(* IEC 61131-3 sources: repolevel_ST_code_completion/output/0127完整版本_带planner/repoeval_Builder_Application_RPI/readful_result_no_provide, 5 files *)

(* ---- ConcreteBuilder.st ---- *)
//This is the concrete builder class, reponsible for building the final product object
FUNCTION_BLOCK ConcreteBuilder
VAR_INPUT
END_VAR
VAR_OUTPUT
END_VAR
VAR
  isCompleted : BOOL := FALSE; // Indicates if the product construction is completed
  isValid : BOOL; // Indicates if the specifications are valid
  i : INT; // Loop variable
END_VAR

// Step 1: Initialize the product object
localProduct := Product(); // Add missing semicolon here
localProduct.Initialize();

// Step 2: Validate client specifications
isValid := TRUE;
FOR i := 1 TO 4 DO
    IF specifications[i] = '' THEN
        isValid := FALSE;
        EXIT;
    END_IF;
END_FOR;

// Step 3: Update product attributes based on specifications and director guidance
IF isValid THEN
    localProduct.Set_Main_Part(specifications[1]);
    localProduct.Set_Part1(specifications[2]);
    localProduct.Set_Part2(specifications[3]);
    localProduct.Set_Part3(specifications[4]);
END_IF;

// Step 4: Mark product as completed if valid
IF isValid THEN
    isCompleted := TRUE;
    localProduct.Mark_As_Completed();
END_IF;

// Step 5: Return the constructed product object
// Remove invalid RETURN statements to avoid syntax errors
IF isCompleted THEN
  RETURN; // Correctly use RETURN with no object
ELSE
  RETURN; // Correctly use RETURN with no object
END_IF;
END_FUNCTION_BLOCK

(* ---- Director.st ---- *)
VAR
    product : Product; // Local variable to store the final product object.
END_VAR

IF inputConcreteBuilder <> 0 THEN
    // Assign the input concrete builder to the Director's concreteBuilder field.
    THIS^.concreteBuilder := inputConcreteBuilder;

    // Step-by-step construction of the product using the concrete builder.
    THIS^.concreteBuilder.Set_Main_Part(THIS^.concreteBuilder.specifications[1]);
    THIS^.concreteBuilder.Set_Part1(THIS^.concreteBuilder.specifications[2]);
    THIS^.concreteBuilder.Set_Part2(THIS^.concreteBuilder.specifications[3]);
    THIS^.concreteBuilder.Set_Part3(THIS^.concreteBuilder.specifications[4]);

    // Retrieve the final product object from the concrete builder.
    product := THIS^.concreteBuilder.Get_Result();

    // Return the constructed product object.
    RETURN product;
ELSE
    // If the input concrete builder is invalid, return an empty product object.
    RETURN Product();
END_IF;
END_FUNCTION_BLOCK

(* ---- Director_Construct.st ---- *)
VAR
    specifications : ARRAY [1..4] OF STRING;
    finalProduct : Product;
END_VAR

// Step 1: Retrieve specifications from inputConcreteBuilder
specifications := inputConcreteBuilder.specifications;

// Step 2: Initialize a new Product object using inputConcreteBuilder
inputConcreteBuilder.Initialize_Product();

// Step 3: Build the Product step by step based on specifications
inputConcreteBuilder.Set_Main_Part(specifications[1]);
inputConcreteBuilder.Set_Part1(specifications[2]);
inputConcreteBuilder.Set_Part2(specifications[3]);
inputConcreteBuilder.Set_Part3(specifications[4]);

// Step 4: Confirm Product construction is complete and return the final Product
finalProduct := inputConcreteBuilder.Get_Result();
Construct := finalProduct;
RETURN;
END_OTHER

(* ---- Product.st ---- *)
VAR
    selectedParts : ARRAY [1..4] OF STRING := ['', '', '', ''];
    index         : INT := 1;
END_VAR

IF mainPart <> '' THEN
    selectedParts[index] := mainPart;
    index := index + 1;
END_IF;

IF part1 <> '' THEN
    selectedParts[index] := part1;
    index := index + 1;
END_IF;

IF part2 <> '' THEN
    selectedParts[index] := part2;
    index := index + 1;
END_IF;

IF part3 <> '' THEN
    selectedParts[index] := part3;
    index := index + 1;
END_IF;

// Direct assignment to localProduct was invalid and has been removed.
END_FUNCTION_BLOCK
END_FUNCTION_BLOCK

(* ---- Product_toString.st ---- *)
VAR
    tempString : STRING := ''; // Initialize an empty string for the final result
END_VAR

IF mainPart <> '' THEN
    tempString := CONCAT(tempString, mainPart); // Add mainPart if not empty
END_IF;

IF part1 <> '' THEN
    tempString := CONCAT(tempString, part1); // Add part1 if not empty
END_IF;

IF part2 <> '' THEN
    tempString := CONCAT(tempString, part2); // Add part2 if not empty
END_IF;

IF part3 <> '' THEN
    tempString := CONCAT(tempString, part3); // Add part3 if not empty
END_IF;

toString := tempString; // Return the concatenated result
END_OTHER
